// Copyright (c) 2024 Loupe (https://loupe.team), provided under the MIT License.

INTERFACE IPLCopenFull EXTENDS __SYSTEM.IQueryInterface


METHOD Aborted : BOOL
VAR_INPUT
END_VAR
END_METHOD


METHOD AbortPreviousCommands : BOOL
VAR_INPUT
  newCommand : IPLCopenCommand;
END_VAR
END_METHOD


PROPERTY Consume : BOOL
GET
END_GET
END_PROPERTY


METHOD Errored : BOOL
VAR_INPUT
  ID : INT;
END_VAR
END_METHOD


PROPERTY Execute : BOOL
SET
END_SET
END_PROPERTY


METHOD Finished : BOOL
VAR_INPUT
END_VAR
END_METHOD


METHOD RegisterGroup : BOOL
VAR_INPUT
  group : IPLCopenGroup;
END_VAR
END_METHOD


{warning 'add property implementation'}
PROPERTY Remote : IPLCopenCallRemote
GET
END_GET
SET
END_SET
END_PROPERTY


PROPERTY Status : PLCopenStatusBase
GET
END_GET
END_PROPERTY

END_INTERFACE

(* stored: Version 1.1.0.1
   Itf IPLCopenFull: Id {c945fc30-fb9b-4180-8aeb-34da6438a603}
   Method Aborted: Id {1bb8dd08-1d55-4829-959e-f4ce3c4cd0fe}
   Method AbortPreviousCommands: Id {245fb2dc-42d2-4fca-ae32-bde199139c9d}
   Property Consume: Id {00a81ccd-7f51-475f-a8fa-00b668582e9c}
   Get Get: Id {76ddde10-39d4-4105-9faf-6c6b895ba3fe}
   Method Errored: Id {893b6b7d-d8dd-4a80-b43e-f2dd179139f3}
   Property Execute: Id {6fe6ce42-a32b-4b6d-8247-cca40e9a3304}
   Set Set: Id {6631e843-65e0-401d-8d1c-2d28f2e296ef}
   Method Finished: Id {1c3d17fa-f354-435f-ab9c-3c1ade19aab4}
   Method RegisterGroup: Id {07f768ee-4e77-40c8-990b-b3741dfe2a7b}
   Property Remote: Id {c789e510-952f-453d-8fde-71b37472057c}
   Get Get: Id {78c5cd67-a3cc-46de-8abd-939e6647b9b6}
   Set Set: Id {fe355a49-1914-427f-879a-8400bdae8f0c}
   Property Status: Id {1e79056e-4c8a-4fbc-a748-d035d0d7e5c2}
   Get Get: Id {d9cfa6b1-6756-4410-91ca-c8981f867a1a} *)
